(* IEC 61131-3 sources: volt/packages/volt-lsp-iec/test-corpus/CodesysTestProject/Device/Plc Logic/Application/Library Manager/IecSfc, 12 files *)

(* ---- SFCACTIONTYPE.dut ---- *)
TYPE SFCACTIONTYPE :
STRUCT
	X : BOOL;
	_X : BOOL;
	T : TIME;
	_T : TIME;
	AC : SFCActionControl;
END_STRUCT
END_TYPE

(* ---- SFCSTEPTYPE.dut ---- *)
TYPE SFCSTEPTYPE :
STRUCT
	X : BOOL;
	T : TIME;
	_X : BOOL;
	_T : TIME;
END_STRUCT
END_TYPE

(* ---- GLOBALE_VARIABLEN.gvl ---- *)
VAR_GLOBAL
END_VAR

(* ---- ISFCELEMENT.itf ---- *)
INTERFACE ISFCELEMENT
END_INTERFACE

METHOD GETPOSTELEMENTS : BOOL
VAR_OUTPUT
	PITFPOSTELEMENTS : POINTER TO ARRAY [0..0] OF ISFCElement;
	UINUMELEMENTS : UINT;
END_VAR
END_METHOD

METHOD GETPREELEMENTS : BOOL
VAR_OUTPUT
	PITFPREELEMENTS : POINTER TO ARRAY [0..0] OF ISFCElement;
	UINUMELEMENTS : UINT;
END_VAR
END_METHOD

(* ---- ISFCJUMP.itf ---- *)
INTERFACE ISFCJUMP
END_INTERFACE

(* ---- ISFCSTEP.itf ---- *)
INTERFACE ISFCSTEP
END_INTERFACE

(* ---- ISFCTRANSITION.itf ---- *)
INTERFACE ISFCTRANSITION
END_INTERFACE

(* ---- SFCACTIONCONTROL.pou ---- *)
FUNCTION_BLOCK SFCACTIONCONTROL
VAR_INPUT
	N : BOOL;
	R0 : BOOL;
	S0 : BOOL;
	L : BOOL;
	D : BOOL;
	P : BOOL;
	SD : BOOL;
	DS : BOOL;
	SL : BOOL;
	T : TIME;
END_VAR
VAR_OUTPUT
	Q : BOOL;
END_VAR
VAR
	S_FF : RS;
	L_TMR : TON;
	D_TMR : TON;
	P_TRIG : R_TRIG;
	SD_TMR : TON;
	SD_FF : RS;
	DS_FF : RS;
	DS_TMR : TON;
	SL_FF : RS;
	SL_TMR : TON;
END_VAR
END_FUNCTION_BLOCK

METHOD RESET
END_METHOD

(* ---- SFCELEMENT.pou ---- *)
FUNCTION_BLOCK SFCELEMENT
VAR_INPUT
	WSNAME : WSTRING;
	PAPREELEMENTS : POINTER TO ARRAY [0..0] OF ISFCElement;
	UIPREELEMENTS : UINT;
	PAPOSTELEMENTS : POINTER TO ARRAY [0..0] OF ISFCElement;
	UIPOSTELEMENTS : UINT;
END_VAR
VAR
	NAME : WSTRING;
END_VAR
END_FUNCTION_BLOCK

METHOD GETPOSTELEMENTS : BOOL
VAR_OUTPUT
	PITFPOSTELEMENTS : POINTER TO ARRAY [0..0] OF ISFCElement;
	UINUMELEMENTS : UINT;
END_VAR
END_METHOD

METHOD GETPREELEMENTS : BOOL
VAR_OUTPUT
	PITFPREELEMENTS : POINTER TO ARRAY [0..0] OF ISFCElement;
	UINUMELEMENTS : UINT;
END_VAR
END_METHOD

(* ---- SFCJUMP.pou ---- *)
FUNCTION_BLOCK SFCJUMP EXTENDS SFCElement
VAR
	ITFSTEP : ISFCStep;
END_VAR
END_FUNCTION_BLOCK

(* ---- SFCSTEP.pou ---- *)
FUNCTION_BLOCK SFCSTEP EXTENDS SFCElement
VAR
	PST : POINTER TO SFCStepType;
	STEPDATA : POINTER TO SFCStepType;
END_VAR
END_FUNCTION_BLOCK

(* ---- SFCTRANSITION.pou ---- *)
FUNCTION_BLOCK SFCTRANSITION EXTENDS SFCElement
VAR
	PBVALUE : POINTER TO BOOL;
	TRANSITIONVALUE : BOOL;
END_VAR
END_FUNCTION_BLOCK
